{attribute 'linkalways'} 
{attribute 'no_explicit_call' := 'This FB is a CLASS and must be accessed using methods or properties'}
{attribute 'enable_dynamic_creation'}
FUNCTION_BLOCK Node_F_VN_AddToContainerElements_TcVnVector4_SINT EXTENDS VisionNode
VAR
    aValue : _TcVnVector4_SINT;
    ipContainer : _ITcVnContainer;
    hrPrev : _HRESULT(S_OK);
    hresult : _HRESULT(S_OK);
END_VAR

METHOD PUBLIC  Clone : I_Node
VAR
    pNode : POINTER TO Node_F_VN_AddToContainerElements_TcVnVector4_SINT;
END_VAR
pNode := __NEW(Node_F_VN_AddToContainerElements_TcVnVector4_SINT);
Clone := pNode^;
END_METHOD

METHOD FB_init : BOOL
VAR_INPUT
    bInitRetains : BOOL; // if TRUE, the retain variables are initialized (warm start / cold start)
    bInCopyCode : BOOL;  // if TRUE, the instance afterwards gets moved into the copy code (online change)
END_VAR
AddInput('aValue', aValue);
AddInput('ipContainer', ipContainer);
AddInput('hrPrev', hrPrev);
AddOutput('ipContainer', ipContainer);
AddOutput('hresult',hresult);
END_METHOD

METHOD PROTECTED OnExecute
hresult.Value := F_VN_AddToContainerElements_TcVnVector4_SINT(
    aValue := aValue.Value,
    ipContainer := ipContainer.Value,
    hrPrev:= hrPrev.Value);
END_METHOD

METHOD PUBLIC PreExecutionCheck
VAR_INPUT
    Check : I_PreExecutionChecks;
END_VAR
Check.IsTrue(ipContainer.IsValid, 'ipContainer must be a valid container');
Check.IsTrue(ipContainer.IsType(TC_GLOBAL_CONST_LIST.ContainerType_Vector_TcVnVector4_SINT), 'ipContainer contains incorrect type');
END_METHOD

END_FUNCTION_BLOCK

(* stored: Version 1.1.0.1, ProductVersion 3.1.4026.13
   POU Node_F_VN_AddToContainerElements_TcVnVector4_SINT: Id {be2d5156-3846-4c1f-a1f3-72031a52503e}, SpecialFunc None
   Folder Constructor: Id {29413b9e-4264-4bc5-8387-48cd42b2d150}
   Method Clone: Id {7870123e-792e-4907-9d13-b5a88585b03c}
   Method FB_init: Id {e40c053f-fdad-452b-8459-b0d35004ea5e}
   Method OnExecute: Id {8625a0ee-8ab0-4166-ad78-49917c109173}
   Method PreExecutionCheck: Id {8accdfb9-1ece-4869-a246-ce900665ea63} *)
